// Sensor Settings
	fbSensor					: SH_Light.FB_NIKO_P46xx_1Pcs;
	//fbSensor					: SH_Light.FB_NIKO_P46xx_3Pcs;
	bySensorAddr				: BYTE := 1;
	//arrSensorAddr				: ARRAY[1..3] OF BYTE := [7,8,9];
	bInitialize					: BOOL := TRUE;
	stDaliSensorSetup			: ST_DALI_NIKOP46SetupData;
	bInitErr					: BOOL;
	bInitDone					: BOOL;
	//arrInitErr				: ARRAY [1..3] OF BOOL;
	//arrInitDone				: ARRAY [1..3] OF BOOL;
	arrSensorScales				: ARRAY [1..10] OF SH_Light.ST_DALI_SensorScaleMode := [
																						(fMeassureMaxSensor := rMeassure_Zone10, fReadMaxSensor := rRead_Zone10),																																									
																						9(())];
	bCancelHoldTimerOccupancy	: BOOL;
(*	eEventPriorityOccupancy		: E_DALIEventPriority := E_DALIEVENTPRIORITY.Middle;
	nHoldTimerOccupancy			: WORD := 5; // Value in s. 	
	nReportTimerOccupancy		: BYTE := 120; // Value in s, Preset manufacturer value
	nDeadtimeTimerOccupancy		: WORD := 100; // Value in ms, Predefined Value of DALI Standard
	bCancelHoldTimerOccupancy	: BOOL;
	nSensitivityOccupancy		: BYTE:= 3; //setting Sensivity (0..4) 0 (Off), 1 (Min), 2(Low), 3(High) and 4 (Max)

	bEnableLuxEvent				: BOOL;
	eEventPriorityBrightness	: E_DALIEventPriority := E_DALIEVENTPRIORITY.Middle;
	nDeadtimeTimerBrightness	: WORD := 1500; // Value in ms, Predefined Value of DALI Standard
	nHysteresisBrightness		: BYTE := 2; // Value in %
	nHysteresisMinBrightness	: BYTE := 10; // Absolute Value, depending on the manufacturer specific resolution
	nReportTimerBrightness		: BYTE := 120; // Value in s, Preset manufacturer value
*)

	//stDaliSetup: SH_Light.ST_DALI_RoomSetup
	//stRoomDataModbus			: SH_Light.ST_RoomDataModbus := ( bPirActive := bPirActive
	

	//ModbusComm setup
	
	fbWriteSPLuxLevel			: SH_Light.FB_TwoVal_SelectOne_RTrigChange;
	fbWritePirDelayTIme		: SH_Light.FB_TwoVal_SelectOne_RTrigChange;
	stRoomDataPLC				: SH_Light.ST_RoomDataPLC	:=	(
																	uiPirOffDelayTime	:= 30,
																	uiSpLuxLevel		:= 500,
																	uiPirDimDelayTime	:= 15,
																	uiSpDimLuxLevel		:= 200);
																	
	fbBallastOnHours				: SH_Light.FB_CountOnHours;
	bEnableHourCount			: BOOL := TRUE;
	
	//Non-persistent modbus data
	bPirActive_MB					AT %MX522.0	: BOOL;				//bPirLys i gammel kode
	uiActLuxLevel_MB			    AT %MB526	: UINT;				//intHMIAktueltLux i gammel kode
	uiActLightLevelPct_MB	        AT %MB530	: UINT;				//intDALI_Gruppe1_Lysniveau i gammel kode
	
	//For Conversion
	uiPirOffMinutes						: UINT;
	udTimeScaling						: UDINT := 60000;
	uiLuxOn								: UINT;
	
	//max values checks
	uiMaxLuxLevel						: UINT := 1023;
	uiMaxPirOffMinutes				    : UINT := 180;

	
END_VAR

VAR CONSTANT
    Sensor_DALI_LINE_NUM				: BYTE := 5;
	DALI_LINE_NUM_LIGHT			     	: BYTE := 2;
	DALI_LINE_NUM_PENDANTS	            : BYTE := 0; //0=ingen pendler	
END_VAR
VAR PERSISTENT
	stPirSensorData: SH_Light.ST_DALI_Sensor;
	stTuneData: SH_Light.ST_TuneData_EX;

	uiPirOffDelayTime_MB	AT %MB524	: UINT;				//ntHMI_Pir_SetValue i gammel kode
	uiSPLuxLevel_MB			AT %MB528	: UINT;				//intHMI_Lux_SetValue i gammel kode
	uiBallastOnHours_MB		AT %MB532	: UINT;				//dintHMILysbraendtimer1 i gammel kode
	byOnHoursOverflowCount				: BYTE;   
END_VAR

A_Buttons();
A_LightCtrl();
A_Sensor();
A_ModbusComm();

ACTION A_Buttons:
bTopButtonZone1		:= bTopButtonZone1_Visu;
bBottomButtonZone1	:= bBottomButtonZone1_Visu;
END_ACTION

ACTION A_LightCtrl:

fbLys(
	nZoneID:= 1, 
	bButtonZone1:= bTopButtonZone1,
	bBottomButtonZone1 := bBottomButtonZone1, 
	//bButtonZone2:= bButtonZone2,
	fLuxOn:= fLuxOn, 
	fLuxDim:= fLuxDim, 
	tPIRDim:= tPIRDim, 
	tPIROff:= tPIROff, 
	fOffsetSec:= fOffsetSec, 
	bReInit:= , 
	stDaliSetup:= stDaliSetup, 
	ipCommunication_Prim:= P_DALI_Background.arrfbKL6821Communication[DALI_LINE_NUM_LIGHT], 
	//ipCommunication_Sec:= P_DALI_Background.arrfbKL6821Communication[DALI_LINE_NUM_LIGHT], 
	//ipCommunication_Supl:= P_DALI_Background.arrfbKL6821Communication[DALI_LINE_NUM_PENDANTS], 
	fMinOutputPowerLevelRoom:= 15, 
	fMaxOutputPowerLevelRoom:= 100, 
	nCycleTimeInMS:= SH_Light.DALI_Param.nPlcTaskCycleTimeInMS*nDimCmdCycleTimeFactor , 
	bRunTuning:= bRunTuning, 
	bOccupiedRoom=> bOccupiedRoom, 
	bError_Prim=> , 
	nError_Prim=> , 
	stTuneData:=stTuneData , 
	stPirSensorData:= stPirSensorData, 
	stLiveData:= stLiveData);
END_ACTION

ACTION A_ModbusComm:
//Manage data for modbus communication

//Manage data for read-only in PLC
stRoomDataPLC.bPirActive			:= stPirSensorData.bPrc;
stRoomDataPLC.uiActLuxLevel			:= TO_UINT(TRUNC(stPirSensorData.fBrightness));
stRoomDataPLC.uiActLightLevelPct	:= TO_UINT(TRUNC(fbLys.fbBallast.fActlLgtLvl_Prim));
		//stRoomDataPLC.uiActLightLevelPct	:= TO_UINT(TRUNC(fbLys.fbBallast.fActlLgtLvl_Prim)); //if only one group light control
stRoomDataPLC.uiBallastOnHours		:= uiBallastOnHours_MB; //The calculation for BallastOnHours is stored directly to the MB register below


//Assign data for read-only to MB registers
bPirActive_MB			:= stRoomDataPLC.bPirActive;
uiActLuxLevel_MB		:= stRoomDataPLC.uiActLuxLevel;
uiActLightLevelPct_MB	:= stRoomDataPLC.uiActLightLevelPct;

	//calculate BallastOnHours
	fbBallastOnHours(
		bEnableHourCount	:= bEnableHourCount,
		bPauseCount			:= fbLys.fbLightCtrl.bOffZone1,
		uiOnHours			:= uiBallastOnHours_MB,			//OnHours is updated here
		byOverflowCount		:= byOnHoursOverflowCount);


//Manage data for read/write for both PLC and MB registers
fbWriteSPLuxLevel(	nMaxValOut	:= uiMaxLuxLevel,
					nValIn1		:= uiSPLuxLevel_MB,		//nValIn1 takes priotity in case of download or restart
					nValIn2		:= stRoomDataPLC.uiSpLuxLevel,
					nValOut		=> uiLuxOn
				);


fbWritePirDelayTIme(	nMaxValOut	:= uiMaxPirOffMinutes,
						nValIn1		:= uiPirOffDelayTime_MB,		//nValIn1 takes priotity in case of download or restart
						nValIn2		:= stRoomDataPLC.uiPirOffDelayTime,
						nValOut		=> uiPirOffMinutes
					);
					

//Convert read/write modbus data to appropriate datatypes in PLC
fLuxOn	:= TO_REAL(uiLuxOn);			
tPIROff	:= TO_TIME(uiPirOffMinutes*udTimeScaling); //Time conversion defaults to ms

fLuxDim	:= TO_REAL(stRoomDataPLC.uiSpDimLuxLevel);			
tPIRDim	:= TO_TIME(stRoomDataPLC.uiPirDimDelayTime*udTimeScaling); //Time conversion defaults to ms
END_ACTION

ACTION A_Sensor:

fbSensor.ipCommunication := P_DALI_Background.arrfbKL6821Communication[Sensor_DALI_LINE_NUM];

//only 1 sensor
fbSensor(
	byShrtAdr:= bySensorAddr,
	bInitialize:= bInitialize, 
	DALI_LINE_NUM:= Sensor_DALI_LINE_NUM, 
 	//bCancelHoldTimerOccupancy:= bCancelHoldTimerOccupancy, 
	stSensorSetup := stDaliSensorSetup,
	bInitErr=> bInitErr, 
	bInitDone=> bInitDone,
	stPirSensorData:= stPirSensorData, 
	arrSensorScales:= arrSensorScales);


(*//several sensors	
fbSensor(
	arrShrtAdr:= arrSensorAddr,
	bInitialize:= bInitialize, 
	DALI_LINE_NUM:= Sensor_DALI_LINE_NUM, 
 	//bCancelHoldTimerOccupancy:= bCancelHoldTimerOccupancy, 
	stSensorSetup := stDaliSensorSetup,
	arrInitErr=> arrInitErr, 
	arrInitDone=> arrInitDone,
	stPirSensorData:= stPirSensorData, 
	arrSensorScales:= arrSensorScales);
	*)
END_ACTION

END_PROGRAM

// ---- POUs/Alle_Rum/Gange/Gang_3_159A_toilet/P_Gang_3_159A.TcPOU
PROGRAM P_Gang_3_159A
VAR

	fbLys		: FB_Light_Type_B;
	

	stDaliSetup	: SH_Light.ST_DALI_RoomSetup := (
														byShrtAdr_Prim := 1, 
														byGrpAdr_Prim := 6,  /////remember
														eMod_Prim := E_DALIAddressType.Group, 
														//byShrtAdr_Sec := 1, 
														//byGrpAdr_Sec := 1, 
														//eMod_Sec := E_DALIAddressType.Short, 
														//byShrtAdr_Supl := 1, 
														DALI_LINE_NUM_PRIM := DALI_LINE_NUM_LIGHT,
														DALI_LINE_NUM_SEC := 0, //0 = ingen zonestyring/vinduerække
													    DALI_LINE_NUM_SUPL := DALI_LINE_NUM_PENDANTS);
														
	stLiveData				: SH_Light.ST_LiveData;
	bRunTuning					: BOOL;
	
	bTopButtonZone1				: BOOL;
	bTopButtonZone1_Visu		: BOOL;
	bBottomButtonZone1			: BOOL;
	bBottomButtonZone1_Visu	    : BOOL;
	bButtonZone2				: BOOL;
	bNeighborRoomsPir			: BOOL;
	fLuxOn						: REAL;
	fLuxDim						: REAL;
	tPIRDim						: TIME;
	tPIROff						: TIME;
	fOffsetSec					: REAL := 20;
	bOccupiedRoom				: BOOL;;


// Sensor Settings
	//fbSensor						: SH_Light.FB_NIKO_P46xx_1Pcs;
	fbSensor						: SH_Light.FB_NIKO_P46xx_2Pcs;
	//bySensorAddr				: BYTE := 1;
	arrSensorAddr				: ARRAY[1..2] OF BYTE := [4,5];
	bInitialize						: BOOL := TRUE;
	stDaliSensorSetup			: ST_DALI_NIKOP46SetupData := (
																nSensitivityPIRSegmentA := arrSensitivityOccupancy[1],
																nSensitivityPIRSegmentB := arrSensitivityOccupancy[2],
																nSensitivityPIRSegmentC := arrSensitivityOccupancy[3]);
	//bInitErr							: BOOL;
	//bInitDone						: BOOL;
	arrInitErr						: ARRAY [1..2] OF BOOL;
	arrInitDone					: ARRAY [1..2] OF BOOL;
	arrSensorScales				: ARRAY [1..10] OF SH_Light.ST_DALI_SensorScaleMode := [
																						(fMeassureMaxSensor := rMeassure_Zone10, fReadMaxSensor := rRead_Zone10),
																						(fMeassureMaxSensor := rMeassure_Zone10, fReadMaxSensor := rRead_Zone10),																																								
																						8(())];
																						
	bCancelHoldTimerOccupancy	: BOOL;
(*	eEventPriorityOccupancy		: E_DALIEventPriority := E_DALIEVENTPRIORITY.Middle;
	nHoldTimerOccupancy			: WORD := 5; // Value in s. 	
	nReportTimerOccupancy		: BYTE := 120; // Value in s, Preset manufacturer value
	nDeadtimeTimerOccupancy		: WORD := 100; // Value in ms, Predefined Value of DALI Standard
	bCancelHoldTimerOccupancy	: BOOL;
	nSensitivityOccupancy		: BYTE:= 3; //setting Sensivity (0..4) 0 (Off), 1 (Min), 2(Low), 3(High) and 4 (Max)

	bEnableLuxEvent				: BOOL;
	eEventPriorityBrightness	: E_DALIEventPriority := E_DALIEVENTPRIORITY.Middle;
	nDeadtimeTimerBrightness	: WORD := 1500; // Value in ms, Predefined Value of DALI Standard
	nHysteresisBrightness		: BYTE := 2; // Value in %
	nHysteresisMinBrightness	: BYTE := 10; // Absolute Value, depending on the manufacturer specific resolution
	nReportTimerBrightness		: BYTE := 120; // Value in s, Preset manufacturer value
*)
	

	//ModbusComm setup
	
	fbWriteSPLuxLevel				: SH_Light.FB_TwoVal_SelectOne_RTrigChange;
	fbWritePirDelayTIme			: SH_Light.FB_TwoVal_SelectOne_RTrigChange;
	stRoomDataPLC					: SH_Light.ST_RoomDataPLC	:=	(
																	uiPirOffDelayTime	:= 30,
																	uiSpLuxLevel			:= 500,
																	uiPirDimDelayTime	:= 15,
																	uiSpDimLuxLevel		:= 200);
																	
	fbBallastOnHours				: SH_Light.FB_CountOnHours;
	bEnableHourCount			: BOOL := TRUE;
	
	//Non-persistent modbus data
	bPirActive_MB				AT %MX534.0	: BOOL;				//bPirLys i gammel kode
	uiActLuxLevel_MB			AT %MB538	: UINT;				//intHMIAktueltLux i gammel kode
	uiActLightLevelPct_MB	    AT %MB542	: UINT;				//intDALI_Gruppe1_Lysniveau i gammel kode
	
	//For Conversion
	uiPirOffMinutes						: UINT;
	udTimeScaling						: UDINT := 60000;
	uiLuxOn								: UINT;
	
	//max values checks
	uiMaxLuxLevel						: UINT := 1023;
	uiMaxPirOffMinutes			    	: UINT := 180;

	
END_VAR

VAR CONSTANT
    Sensor_DALI_LINE_NUM				: BYTE := 4;
	DALI_LINE_NUM_LIGHT			    	: BYTE := 4;
	DALI_LINE_NUM_PENDANTS	            : BYTE := 0; //0=ingen pendler
	arrSensitivityOccupancy						: ARRAY[1..3] OF BYTE := [4,4,4];
END_VAR
VAR PERSISTENT
	stPirSensorData: SH_Light.ST_DALI_Sensor;
	stTuneData: SH_Light.ST_TuneData_EX;

	uiPirOffDelayTime_MB	AT %MB536	: UINT;				//ntHMI_Pir_SetValue i gammel kode
	uiSPLuxLevel_MB			AT %MB540	: UINT;				//intHMI_Lux_SetValue i gammel kode
	uiBallastOnHours_MB		AT %MB544	: UINT;				//dintHMILysbraendtimer1 i gammel kode
	byOnHoursOverflowCount							: BYTE;   
END_VAR

A_Buttons();
A_LightCtrl();
A_Sensor();
A_ModbusComm();

ACTION A_Buttons:
bTopButtonZone1		:= bTopButtonZone1_Visu;
bBottomButtonZone1	:= bBottomButtonZone1_Visu;
END_ACTION

ACTION A_LightCtrl:

fbLys(
	nZoneID:= 1, 
	bButtonZone1:= bTopButtonZone1,
	bBottomButtonZone1 := bBottomButtonZone1, 
	//bButtonZone2:= bButtonZone2, 
	bNeighborRoomsPir	:=	bNeighborRoomsPir,
	fLuxOn:= fLuxOn, 
	fLuxDim:= fLuxDim, 
	tPIRDim:= tPIRDim, 
	tPIROff:= tPIROff, 
	fOffsetSec:= fOffsetSec, 
	bReInit:= , 
	stDaliSetup:= stDaliSetup, 
	ipCommunication_Prim:= P_DALI_Background.arrfbKL6821Communication[DALI_LINE_NUM_LIGHT], 
	//ipCommunication_Sec:= P_DALI_Background.arrfbKL6821Communication[DALI_LINE_NUM_LIGHT], 
	//ipCommunication_Supl:= P_DALI_Background.arrfbKL6821Communication[DALI_LINE_NUM_PENDANTS], 
	fMinOutputPowerLevelRoom:= 15, 
	fMaxOutputPowerLevelRoom:= 100, 
	nCycleTimeInMS:= SH_Light.DALI_Param.nPlcTaskCycleTimeInMS*nDimCmdCycleTimeFactor , 
	bRunTuning:= bRunTuning, 
	bOccupiedRoom=> bOccupiedRoom, 
	bError_Prim=> , 
	nError_Prim=> , 
	stTuneData:=stTuneData , 
	stPirSensorData:= stPirSensorData, 
	stLiveData:= stLiveData);
END_ACTION

ACTION A_ModbusComm:
//Manage data for modbus communication

//Manage data for read-only in PLC
stRoomDataPLC.bPirActive			:= stPirSensorData.bPrc;
stRoomDataPLC.uiActLuxLevel			:= TO_UINT(TRUNC(stPirSensorData.fBrightness));
stRoomDataPLC.uiActLightLevelPct	:= TO_UINT(TRUNC(fbLys.fbBallast.fActlLgtLvl_Prim));
		//stRoomDataPLC.uiActLightLevelPct	:= TO_UINT(TRUNC(fbLys.fbBallast.fActlLgtLvl_Prim)); //if only one group light control
stRoomDataPLC.uiBallastOnHours		:= uiBallastOnHours_MB; //The calculation for BallastOnHours is stored directly to the MB register below


//Assign data for read-only to MB registers
bPirActive_MB			:= stRoomDataPLC.bPirActive;
uiActLuxLevel_MB		:= stRoomDataPLC.uiActLuxLevel;
uiActLightLevelPct_MB	:= stRoomDataPLC.uiActLightLevelPct;

	//calculate BallastOnHours
	fbBallastOnHours(
		bEnableHourCount	:= bEnableHourCount,
		bPauseCount			:= fbLys.fbLightCtrl.bOffZone1,
		uiOnHours			:= uiBallastOnHours_MB,			//OnHours is updated here
		byOverflowCount		:= byOnHoursOverflowCount);


//Manage data for read/write for both PLC and MB registers
fbWriteSPLuxLevel(	nMaxValOut	:= uiMaxLuxLevel,
					nValIn1		:= uiSPLuxLevel_MB,		//nValIn1 takes priotity in case of download or restart
					nValIn2		:= stRoomDataPLC.uiSpLuxLevel,
					nValOut		=> uiLuxOn
				);


fbWritePirDelayTIme(	nMaxValOut	:= uiMaxPirOffMinutes,
						nValIn1		:= uiPirOffDelayTime_MB,		//nValIn1 takes priotity in case of download or restart
						nValIn2		:= stRoomDataPLC.uiPirOffDelayTime,
						nValOut		=> uiPirOffMinutes
					);
					

//Convert read/write modbus data to appropriate datatypes in PLC
fLuxOn	:= TO_REAL(uiLuxOn);			
tPIROff	:= TO_TIME(uiPirOffMinutes*udTimeScaling); //Time conversion defaults to ms

fLuxDim	:= TO_REAL(stRoomDataPLC.uiSpDimLuxLevel);			
tPIRDim	:= TO_TIME(stRoomDataPLC.uiPirDimDelayTime*udTimeScaling); //Time conversion defaults to ms
END_ACTION

ACTION A_Sensor:

fbSensor.ipCommunication := P_DALI_Background.arrfbKL6821Communication[Sensor_DALI_LINE_NUM];

//only 1 sensor
(*fbSensor(
	byShrtAdr:= bySensorAddr,
	bInitialize:= bInitialize, 
	DALI_LINE_NUM:= Sensor_DALI_LINE_NUM, 
 	//bCancelHoldTimerOccupancy:= bCancelHoldTimerOccupancy, 
	stSensorSetup := stDaliSensorSetup,
	bInitErr=> bInitErr, 
	bInitDone=> bInitDone,
	stPirSensorData:= stPirSensorData, 
	arrSensorScales:= arrSensorScales);
*)

//several sensors	
fbSensor(
	arrShrtAdr:= arrSensorAddr,
	bInitialize:= bInitialize, 
	DALI_LINE_NUM:= Sensor_DALI_LINE_NUM, 
 	//bCancelHoldTimerOccupancy:= bCancelHoldTimerOccupancy, 
	stSensorSetup := stDaliSensorSetup,
	arrInitErr=> arrInitErr, 
	arrInitDone=> arrInitDone,
	stPirSensorData:= stPirSensorData, 
	arrSensorScales:= arrSensorScales);
END_ACTION

END_PROGRAM

// ---- POUs/Alle_Rum/Trapper/P_Trappe_T2.TcPOU
PROGRAM P_Trappe_T2
VAR
	bDigitalPir				AT%I*	: BOOL;
	bTrappelysNC		AT%Q*	: BOOL;
	

		
		
	fbTon_Off				: TON;
	tPirTidOff				: TIME;
	tPirTidOff_PLC	: TIME := T#1M;
	bIngenAktivitet		: BOOL;
	bTrappeLys			: BOOL;
	
	//Modbus data Read
	bTrappeAktivitet		: BOOL;
	//Modbus data Read/Wrtite
	bPirTidOff_MB			: TIME;
	
END_VAR


bIngenAktivitet	:= NOT bDigitalPir;
tPirTidOff		:= tPirTidOff_PLC;

fbTon_Off(IN:= bIngenAktivitet, PT:= tPirTidOff);

IF bDigitalPir  THEN
	bTrappeLys := TRUE;
END_IF
IF fbTon_Off.Q THEN
	bTrappeLys := FALSE;
END_IF

bTrappelysNC 	:= NOT bTrappeLys;

END_PROGRAM

// ---- POUs/Alle_Rum/Trapper/P_Trappe_T3.TcPOU
PROGRAM P_Trappe_T3
VAR
	bDigitalPir				AT%I*	: BOOL;
	bTrappelysNC		AT%Q*	: BOOL;
	

		
		
	fbTon_Off				: TON;
	tPirTidOff				: TIME;
	tPirTidOff_PLC	: TIME := T#1M;
	bIngenAktivitet		: BOOL;
	bTrappeLys			: BOOL;
	
	//Modbus data Read
	bTrappeAktivitet		: BOOL;
	//Modbus data Read/Wrtite
	bPirTidOff_MB			: TIME;
	
END_VAR


bIngenAktivitet	:= NOT bDigitalPir;
tPirTidOff		:= tPirTidOff_PLC;

fbTon_Off(IN:= bIngenAktivitet, PT:= tPirTidOff);

IF bDigitalPir  THEN
	bTrappeLys := TRUE;
END_IF
IF fbTon_Off.Q THEN
	bTrappeLys := FALSE;
END_IF

bTrappelysNC 	:= NOT bTrappeLys;

END_PROGRAM

// ---- POUs/DALI/DALI_Setup/FBs/FB_Part202Emergency.TcPOU
FUNCTION_BLOCK FB_Part202Emergency
VAR_INPUT
	ipDALICommunication					:	I_DALICommunication;
END_VAR
VAR_OUTPUT
	bBusy								:	BOOL;
END_VAR
VAR
	{region "Visu"}
	bReadCommands						:	BOOL;
	bReadState							:	BOOL;
	bReadParameter						:	BOOL;
	bStartFunctionTest					:	BOOL;
	bStopTest							:	BOOL;
	bStartDurationTest					:	BOOL;
	bResetFunctionTestDoneFlag			:	BOOL;
	bResetDurationTestDoneFlag			:	BOOL;
	bInhibit							:	BOOL;
	bResetInhibit						:	BOOL;
	bResetLampTime						:	BOOL;
	bRest								:	BOOL;
	bStartIdentification				:	BOOL;
	bWrite								:	BOOL;
	nBatteryCharge						:	BYTE;
	nDurationTestResult					:	BYTE;
	nLampEmergencyTime					:	BYTE;
	nLampTotalOperationTime				:	BYTE;
	sRestMode							:	STRING[5];
	sNormalMode							:	STRING[5];
	sEmergencyMode						:	STRING[5];
	sExtendedEmergency					:	STRING[5];
	sFunctionTest						:	STRING[5];
	sDurationTest						:	STRING[5];
	sHardwiredInhibit					:	STRING[5];
	sHardwiredSwitch					:	STRING[5];

	sCircuitFailure						:	STRING[5];
	sBatteryDurationFailure				:	STRING[5];
	sBatteryFailure						:	STRING[5];
	sEmergencyLampFailure				:	STRING[5];
	sFunctionTestExceed					:	STRING[5];
	sDurationTestExceed					:	STRING[5];
	sFunctionTestFailed					:	STRING[5];
	sDurationTestFailed					:	STRING[5];

	sInhibitMode						:	STRING[5];
	sFunctionTestDoneValid				:	STRING[5];
	sDurationTestDoneValid				:	STRING[5];
	sBatteryFullCharged					:	STRING[5];
	sFunctionTestRequestPending			:	STRING[5];
	sDurationTestRequestPending			:	STRING[5];
	sIdentificationActive				:	STRING[5];

	bIntegralControlGear				:	BOOL;
	bMaintainedControlGear				:	BOOL;
	bSwitchtedMaintainedControlGear		:	BOOL;
	bAutoTestCapability					:	BOOL;
	bAdjustableEmergencyLevel			:	BOOL;
	bHardwiredInhibitSupported			:	BOOL;
	bPhysicalSelectionSupported			:	BOOL;
	bRelightinRestModeSupported			:	BOOL;

	nEmergencyLevel						:	BYTE;
	nEmergencyMinLevel					:	BYTE;
	nEmergencyMaxLevel					:	BYTE;
	nProlongTime						:	UINT;
	fDurationTestDelayTimeVisu			:	REAL;
	fFunctionTestDelayTimeVisu			:	REAL;
	nFunctionTestInterval				:	UINT;
	nDurationTestInterval				:	UINT;
	nTestExecutionTimeout				:	UINT;
	nRatedDuration						:	BYTE;
	{endregion}
	nStep								:	INT;
	nAddress							:	BYTE;
	bHideWaitSymbol						:	BOOL := TRUE;
	
	nDurationTestDelayTime				:	UINT;
	nFunctionTestDelayTime				:	UINT;
	
	fb103StartQuiescentMode				:	FB_DALI103StartQuiescentMode(0);
	fb103StopQuiescentMode				:	FB_DALI103StopQuiescentMode(0);
	fb202QueryBatteryCharge				:	FB_DALI202QueryBatteryCharge(0);
	fb202QueryDurationTestResult		:	FB_DALI202QueryDurationTestResult(0);
	fb202QueryLampEmergencyTime			:	FB_DALI202QueryLampEmergencyTime(0);
	fb202QueryLampTotalOperationTime	:	FB_DALI202QueryLampTotalOperationTime(0);
	fb202QueryEmergencyLevel			:	FB_DALI202QueryEmergencyLevel(0);
	fb202QueryEmergencyMode				:	FB_DALI202QueryEmergencyMode(0);
	fb202QueryFailureStatus				:	FB_DALI202QueryFailureStatus(0);
	fb202QueryEmergencyStatus			:	FB_DALI202QueryEmergencyStatus(0);
	
	fb202QueryEmergencyMinLevel			:	FB_DALI202QueryEmergencyMinLevel(0);
	fb202QueryEmergencyMaxLevel			:	FB_DALI202QueryEmergencyMaxLevel(0);
	fb202QueryTestTiming				:	FB_DALI202QueryTestTiming(0);
	fb202QueryRatedDuration				:	FB_DALI202QueryRatedDuration(0);
	fb202QueryFeatures					:	FB_DALI202QueryFeatures(0);
	
	fb202SetEmergencyLevel				:	FB_DALI202SetEmergencyLevel(0);
	fb202SetProlongTime					:	FB_DALI202SetProlongTime(0);
	fb202SetTestDelayTime				:	FB_DALI202SetTestDelayTime(0);
	fb202SetFunctionTestInterval		:	FB_DALI202SetFunctionTestInterval(0);
	fb202SetDurationTestInterval		:	FB_DALI202SetDurationTestInterval(0);
	fb202SetTestExecutionTimeout		:	FB_DALI202SetTestExecutionTimeout(0);
	
	fb202StartFunctionTest				:	FB_DALI202StartFunctionTest(0);
	fb202StopTest						:	FB_DALI202StopTest(0);
	fb202StartDurationTest				:	FB_DALI202StartDurationTest(0);
	fb202ResetFunctionTestDoneFlag		:	FB_DALI202ResetFunctionTestDoneFlag(0);
	fb202ResetDurationTestDoneFlag		:	FB_DALI202ResetDurationTestDoneFlag(0);
	fb202Inhibit						:	FB_DALI202Inhibit(0);
	fb202ReLightResetInhibit			:	FB_DALI202ReLightResetInhibit(0);
	fb202ResetLampTime					:	FB_DALI202ResetLampTime(0);
	fb202Rest							:	FB_DALI202Rest(0);
	fb202StartIdentification			:	FB_DALI202StartIdentification(0);
END_VAR

{region "Detect Commands"}
IF (bStartFunctionTest AND (nStep = 0)) THEN
	nStep := 5;
	bStartFunctionTest := FALSE;
END_IF

IF (bStopTest AND (nStep = 0)) THEN
	nStep := 10;
	bStopTest := FALSE;
END_IF

IF (bStartDurationTest AND (nStep = 0)) THEN
	nStep := 15;
	bStartDurationTest := FALSE;
END_IF

IF (bResetFunctionTestDoneFlag AND (nStep = 0)) THEN
	nStep := 20;
	bResetFunctionTestDoneFlag := FALSE;
END_IF

IF (bResetDurationTestDoneFlag AND (nStep = 0)) THEN
	nStep := 25;
	bResetDurationTestDoneFlag := FALSE;
END_IF

IF (bInhibit AND (nStep = 0)) THEN
	nStep := 30;
	bInhibit := FALSE;
END_IF

IF (bResetInhibit AND (nStep = 0)) THEN
	nStep := 35;
	bResetInhibit := FALSE;
END_IF

IF (bResetLampTime AND (nStep = 0)) THEN
	nStep := 40;
	bResetLampTime := FALSE;
END_IF			   
					
IF (bRest AND (nStep = 0)) THEN
	nStep := 45;
	bRest := FALSE;
END_IF

IF (bStartIdentification AND (nStep = 0)) THEN
	nStep := 50;
	bStartIdentification := FALSE;
END_IF

IF (bReadCommands AND (nStep = 0)) THEN
	nStep := 60;
	bReadCommands := FALSE;
	bHideWaitSymbol := FALSE;
END_IF

IF (bReadState AND (nStep = 0)) THEN
	nStep := 100;
	bReadState := FALSE;
	bHideWaitSymbol := FALSE;
END_IF

IF (bReadParameter AND (nStep = 0)) THEN
	nStep := 200;
	bReadParameter := FALSE;
	bHideWaitSymbol := FALSE;
END_IF

IF (bWrite AND (nStep = 0)) THEN
	nStep := 500;
	bWrite := FALSE;
	bHideWaitSymbol := FALSE;
END_IF
{endregion}
{region "Manage Dialog Selection}
IF (nStep = 0) THEN
	bBusy := FALSE;
ELSE
	bBusy := TRUE;
END_IF
{endregion}
{region "Execute Commands"}
CASE nStep OF
0:
{region "Init"}
	bReadCommands := FALSE;
	bReadState := FALSE;
	bReadParameter := FALSE;
	bWrite := FALSE;
	bHideWaitSymbol := TRUE;

	fb103StartQuiescentMode.ipDALICommunication := ipDALICommunication;
	fb103StopQuiescentMode.ipDALICommunication := ipDALICommunication;
	fb202QueryBatteryCharge.ipDALICommunication := ipDALICommunication;
	fb202QueryDurationTestResult.ipDALICommunication := ipDALICommunication;
	fb202QueryDurationTestResult.ipDALICommunication := ipDALICommunication;
	fb202QueryLampEmergencyTime.ipDALICommunication := ipDALICommunication;
	fb202QueryLampTotalOperationTime.ipDALICommunication := ipDALICommunication;
	fb202QueryEmergencyMode.ipDALICommunication := ipDALICommunication;
	fb202QueryFailureStatus.ipDALICommunication := ipDALICommunication;
	fb202QueryEmergencyStatus.ipDALICommunication := ipDALICommunication;
	fb202QueryEmergencyLevel.ipDALICommunication := ipDALICommunication;
	fb202QueryEmergencyMinLevel.ipDALICommunication := ipDALICommunication;
	fb202QueryEmergencyMaxLevel.ipDALICommunication := ipDALICommunication;
	fb202QueryTestTiming.ipDALICommunication := ipDALICommunication;
	fb202QueryRatedDuration.ipDALICommunication := ipDALICommunication;
	fb202QueryFeatures.ipDALICommunication := ipDALICommunication;
	fb202SetEmergencyLevel.ipDALICommunication := ipDALICommunication;
	fb202SetProlongTime.ipDALICommunication := ipDALICommunication;
	fb202SetTestDelayTime.ipDALICommunication := ipDALICommunication;
	fb202SetFunctionTestInterval.ipDALICommunication := ipDALICommunication;
	fb202SetDurationTestInterval.ipDALICommunication := ipDALICommunication;
	fb202SetTestExecutionTimeout.ipDALICommunication := ipDALICommunication;

	fb202StartFunctionTest.ipDALICommunication := ipDALICommunication;
	fb202StopTest.ipDALICommunication := ipDALICommunication;
	fb202StartDurationTest.ipDALICommunication := ipDALICommunication;
	fb202ResetFunctionTestDoneFlag.ipDALICommunication := ipDALICommunication;
	fb202ResetDurationTestDoneFlag.ipDALICommunication := ipDALICommunication;
	fb202Inhibit.ipDALICommunication := ipDALICommunication;
	fb202ReLightResetInhibit.ipDALICommunication := ipDALICommunication;
	fb202ResetLampTime.ipDALICommunication := ipDALICommunication;
	fb202Rest.ipDALICommunication := ipDALICommunication;
	fb202StartIdentification.ipDALICommunication := ipDALICommunication;
{endregion}
{region "Commands"}
5:
	fb202StartFunctionTest(	bStart:= TRUE,
							nAddress := nAddress,
							eAddressType := Tc3_DALI.E_DALIAddressType.Short,
							eCommandPriority := Tc3_DALI.E_DALICommandPriority.Middle);
	IF (NOT fb202StartFunctionTest.bBusy) THEN
		fb202StartFunctionTest(bStart := FALSE);
		nStep :=0;
	END_IF
10:
	fb202StopTest(	bStart:= TRUE,
					nAddress := nAddress,
					eAddressType := Tc3_DALI.E_DALIAddressType.Short,
					eCommandPriority := Tc3_DALI.E_DALICommandPriority.Middle);
	IF (NOT fb202StopTest.bBusy) THEN
		fb202StopTest(bStart := FALSE);
		nStep :=0;
	END_IF
15:
	fb202StartDurationTest(	bStart:= TRUE,
							nAddress := nAddress,
							eAddressType := Tc3_DALI.E_DALIAddressType.Short,
							eCommandPriority := Tc3_DALI.E_DALICommandPriority.Middle);
	IF (NOT fb202StartDurationTest.bBusy) THEN
		fb202StartDurationTest(bStart := FALSE);
		nStep := 0;
	END_IF
20:
	fb202ResetFunctionTestDoneFlag(	bStart := TRUE,
									nAddress := nAddress,
									eAddressType := Tc3_DALI.E_DALIAddressType.Short,
									eCommandPriority := Tc3_DALI.E_DALICommandPriority.Middle);
	IF (NOT fb202ResetFunctionTestDoneFlag.bBusy) THEN
		fb202ResetFunctionTestDoneFlag(bStart := FALSE);
		nStep := 0;
	END_IF
25:
	fb202ResetDurationTestDoneFlag(	bStart:= TRUE,
									nAddress := nAddress,
									eAddressType := Tc3_DALI.E_DALIAddressType.Short,
									eCommandPriority := Tc3_DALI.E_DALICommandPriority.Middle);
	IF (NOT fb202ResetDurationTestDoneFlag.bBusy) THEN
		fb202ResetDurationTestDoneFlag(bStart := FALSE);
		nStep := 0;
	END_IF
30:
	fb202Inhibit(	bStart := TRUE,
					nAddress := nAddress,
					eAddressType := Tc3_DALI.E_DALIAddressType.Short,
					eCommandPriority := Tc3_DALI.E_DALICommandPriority.Middle);
	IF (NOT fb202Inhibit.bBusy) THEN
		fb202Inhibit(bStart := FALSE);
		nStep := 0;
	END_IF
35:
	fb202ReLightResetInhibit(	bStart := TRUE,
								nAddress := nAddress,
								eAddressType := Tc3_DALI.E_DALIAddressType.Short,
								eCommandPriority := Tc3_DALI.E_DALICommandPriority.Middle);
	IF (NOT fb202ReLightResetInhibit.bBusy) THEN
		fb202ReLightResetInhibit(bStart := FALSE);
		nStep := 0;
	END_IF
40:
	fb202ResetLampTime(	bStart := TRUE,
						nAddress := nAddress,
						eAddressType := Tc3_DALI.E_DALIAddressType.Short,
						eCommandPriority := Tc3_DALI.E_DALICommandPriority.Middle);
	IF (NOT fb202ResetLampTime.bBusy) THEN
		fb202ResetLampTime(bStart := FALSE);
		nStep := 0;
	END_IF
45:
	fb202Rest(	bStart := TRUE,
				nAddress := nAddress,
				eAddressType := Tc3_DALI.E_DALIAddressType.Short,
				eCommandPriority := Tc3_DALI.E_DALICommandPriority.Middle);
	IF (NOT fb202Rest.bBusy) THEN
		fb202Rest(bStart := FALSE);
		nStep := 0;
	END_IF
50:
	fb202StartIdentification(	bStart := TRUE,
								nAddress := nAddress,
								eAddressType := Tc3_DALI.E_DALIAddressType.Short,
								eCommandPriority := Tc3_DALI.E_DALICommandPriority.Middle);
	IF (NOT fb202StartIdentification.bBusy) THEN
		fb202StartIdentification(bStart := FALSE);
		nStep := 0;
	END_IF
{endregion}
{region "Read Command Status"}
55:
{region "Start Qiescent Mode"}
	fb103StartQuiescentMode(bStart := TRUE,
							eAddressType := Tc3_DALI.E_DALIAddressType.Broadcast,
							eCommandPriority := Tc3_DALI.E_DALICommandPriority.Middle);
	IF (NOT fb103StartQuiescentMode.bBusy) THEN
		fb103StartQuiescentMode(bStart := FALSE);
		nStep := 60;
	END_IF
{endregion}
{endregion}
60:
{region "Query Battery Charge"}
	fb202QueryBatteryCharge(bStart := TRUE,
							nAddress := nAddress,
							eAddressType := Tc3_DALI.E_DALIAddressType.Short,
							eCommandPriority := Tc3_DALI.E_DALICommandPriority.Middle );
	IF (NOT fb202QueryBatteryCharge.bBusy) THEN
		fb202QueryBatteryCharge(bStart:= FALSE);
		nBatteryCharge := fb202QueryBatteryCharge.nBatteryCharge;
		nStep := 65;
	END_IF
{endregion}
65:
{region "Query Duration Test Result"}
	fb202QueryDurationTestResult(	bStart := TRUE,
									nAddress := nAddress,
									eAddressType := Tc3_DALI.E_DALIAddressType.Short,
									eCommandPriority := Tc3_DALI.E_DALICommandPriority.Middle );
	IF (NOT fb202QueryDurationTestResult.bBusy) THEN
		fb202QueryDurationTestResult(bStart := FALSE);
		nDurationTestResult := (2 * fb202QueryDurationTestResult.nDurationTestResult);
		nStep := 70;
	END_IF
{endregion}
70:
{region "Query Lamp emergency Time"}
	fb202QueryLampEmergencyTime(	bStart := TRUE,
									nAddress := nAddress,
									eAddressType := Tc3_DALI.E_DALIAddressType.Short,
									eCommandPriority := Tc3_DALI.E_DALICommandPriority.Middle );
	IF (NOT fb202QueryLampEmergencyTime.bBusy) THEN
		fb202QueryLampEmergencyTime(bStart := FALSE);
		nLampEmergencyTime := fb202QueryLampEmergencyTime.nLampEmergencyTime;
		nStep := 75;
	END_IF
{endregion}
75:
{region "Query Lamp total operation Time"}
	fb202QueryLampTotalOperationTime(	bStart := TRUE,
										nAddress := nAddress,
										eAddressType := Tc3_DALI.E_DALIAddressType.Short,
										eCommandPriority := Tc3_DALI.E_DALICommandPriority.Middle );
	IF (NOT fb202QueryLampTotalOperationTime.bBusy) THEN
		fb202QueryLampTotalOperationTime(bStart:= FALSE);
		nLampTotalOperationTime := (4 * fb202QueryLampTotalOperationTime.nLampTotalOperationTime);
		nStep := 80;
	END_IF
{endregion}
80:
{region "Stop Quiescent Mode"}
	fb103StopQuiescentMode(bStart := TRUE,
							eAddressType := Tc3_DALI.E_DALIAddressType.Broadcast,
							eCommandPriority := Tc3_DALI.E_DALICommandPriority.Middle);
	IF (NOT fb103StopQuiescentMode.bBusy) THEN
		fb103StopQuiescentMode(bStart := FALSE);
		nStep := 0;
	END_IF
	{endregion}

{region "Read Status"}
100:
{region "Query Emergency Mode"}
	fb202QueryEmergencyMode(bStart := TRUE,
							nAddress := nAddress,
							eAddressType := Tc3_DALI.E_DALIAddressType.Short,
							eCommandPriority := Tc3_DALI.E_DALICommandPriority.Middle );
	IF (NOT fb202QueryEmergencyMode.bBusy) THEN
		fb202QueryEmergencyMode(bStart:= FALSE);
		sRestMode := SEL(fb202QueryEmergencyMode.nEmergencyMode.0, 'FALSE', 'TRUE');
		sNormalMode := SEL(fb202QueryEmergencyMode.nEmergencyMode.1, 'FALSE', 'TRUE');
		sEmergencyMode := SEL(fb202QueryEmergencyMode.nEmergencyMode.2, 'FALSE', 'TRUE');
		sExtendedEmergency := SEL(fb202QueryEmergencyMode.nEmergencyMode.3, 'FALSE', 'TRUE');
		sFunctionTest := SEL(fb202QueryEmergencyMode.nEmergencyMode.4, 'FALSE', 'TRUE');
		sDurationTest := SEL(fb202QueryEmergencyMode.nEmergencyMode.5, 'FALSE', 'TRUE');
		sHardwiredInhibit := SEL(fb202QueryEmergencyMode.nEmergencyMode.6, 'FALSE', 'TRUE');
		sHardwiredSwitch := SEL(fb202QueryEmergencyMode.nEmergencyMode.7, 'FALSE', 'TRUE');
		nStep := 110;
	END_IF
{endregion}
110:
{region "Query Failure Status"}
	fb202QueryFailureStatus(bStart := TRUE,
							nAddress := nAddress,
							eAddressType := Tc3_DALI.E_DALIAddressType.Short,
							eCommandPriority := Tc3_DALI.E_DALICommandPriority.Middle );
	IF (NOT fb202QueryFailureStatus.bBusy) THEN
		fb202QueryFailureStatus(bStart := FALSE);
		sCircuitFailure := SEL(fb202QueryFailureStatus.nFailureStatus.0, 'FALSE', 'TRUE');
		sBatteryDurationFailure := SEL(fb202QueryFailureStatus.nFailureStatus.1, 'FALSE', 'TRUE');
		sBatteryFailure := SEL(fb202QueryFailureStatus.nFailureStatus.2, 'FALSE', 'TRUE');
		sEmergencyLampFailure := SEL(fb202QueryFailureStatus.nFailureStatus.3, 'FALSE', 'TRUE');
		sFunctionTestExceed := SEL(fb202QueryFailureStatus.nFailureStatus.4, 'FALSE', 'TRUE');
		sDurationTestExceed := SEL(fb202QueryFailureStatus.nFailureStatus.5, 'FALSE', 'TRUE');
		sFunctionTestFailed := SEL(fb202QueryFailureStatus.nFailureStatus.6, 'FALSE', 'TRUE');
		sDurationTestFailed := SEL(fb202QueryFailureStatus.nFailureStatus.7, 'FALSE', 'TRUE');
		nStep := 120;
	END_IF
{endregion}
120:
{region "Query Emergency Status"}
	fb202QueryEmergencyStatus(bStart := TRUE,
							nAddress := nAddress,
							eAddressType := Tc3_DALI.E_DALIAddressType.Short,
							eCommandPriority := Tc3_DALI.E_DALICommandPriority.Middle );
	IF (NOT fb202QueryEmergencyStatus.bBusy) THEN
		fb202QueryEmergencyStatus(bStart := FALSE);
		sInhibitMode := SEL(fb202QueryEmergencyStatus.nEmergencyStatus.0, 'FALSE', 'TRUE');
		sFunctionTestDoneValid := SEL(fb202QueryEmergencyStatus.nEmergencyStatus.1, 'FALSE', 'TRUE');
		sDurationTestDoneValid := SEL(fb202QueryEmergencyStatus.nEmergencyStatus.2, 'FALSE', 'TRUE');
		sBatteryFullCharged := SEL(fb202QueryEmergencyStatus.nEmergencyStatus.3, 'FALSE', 'TRUE');
		sFunctionTestRequestPending := SEL(fb202QueryEmergencyStatus.nEmergencyStatus.4, 'FALSE', 'TRUE');
		sDurationTestRequestPending := SEL(fb202QueryEmergencyStatus.nEmergencyStatus.5, 'FALSE', 'TRUE');
		sIdentificationActive := SEL(fb202QueryEmergencyStatus.nEmergencyStatus.6, 'FALSE', 'TRUE');
		nStep := 0;
	END_IF
{endregion}
{endregion}
{region "Read Parameters"}
200:
	{region "Start Qiescent Mode"}
	fb103StartQuiescentMode(bStart := TRUE,
							eAddressType := Tc3_DALI.E_DALIAddressType.Broadcast,
							eCommandPriority := Tc3_DALI.E_DALICommandPriority.Middle);
	IF (NOT fb103StartQuiescentMode.bBusy) THEN
		fb103StartQuiescentMode(bStart := FALSE);
		nStep := 210;
	END_IF
{endregion}
210:
{region "Query Emergency Level"}
	fb202QueryEmergencyLevel(	bStart := TRUE,
								nAddress := nAddress,
								eAddressType := Tc3_DALI.E_DALIAddressType.Short,
								eCommandPriority := Tc3_DALI.E_DALICommandPriority.Middle );
	IF (NOT fb202QueryEmergencyLevel.bBusy) THEN
		fb202QueryEmergencyLevel (bStart := FALSE);
		nEmergencyLevel := fb202QueryEmergencyLevel.nEmergencyLevel;
		nStep := 220;
	END_IF
{endregion}
220:
{region "Query Emergency Min Level"}
	fb202QueryEmergencyMinLevel(bStart := TRUE,
								nAddress := nAddress,
								eAddressType := Tc3_DALI.E_DALIAddressType.Short,
								eCommandPriority := Tc3_DALI.E_DALICommandPriority.Middle );
	IF (NOT fb202QueryEmergencyMinLevel.bBusy) THEN
		fb202QueryEmergencyMinLevel (bStart := FALSE);
		nEmergencyMinLevel := fb202QueryEmergencyMinLevel.nEmergencyMinLevel;
		nStep := 230;
	END_IF
{endregion}
230:
{region "Query Emergency Max Level"}
	fb202QueryEmergencyMaxLevel(bStart := TRUE,
								nAddress := nAddress,
								eAddressType := Tc3_DALI.E_DALIAddressType.Short,
								eCommandPriority := Tc3_DALI.E_DALICommandPriority.Middle );
	IF (NOT fb202QueryEmergencyMaxLevel.bBusy) THEN
		fb202QueryEmergencyMaxLevel (bStart := FALSE);
		nEmergencyMaxLevel := fb202QueryEmergencyMaxLevel.nEmergencyMaxLevel;
		nStep := 240;
	END_IF
{endregion}
240: 
{region "Query Prolong Time"}
	fb202QueryTestTiming(	bStart := TRUE,
							nAddress := nAddress,
							eAddressType := Tc3_DALI.E_DALIAddressType.Short,
							eCommandPriority := Tc3_DALI.E_DALICommandPriority.Middle,
							eTestTiming:= Tc3_DALI.E_DALITestTiming.ProlongTime);
	IF (NOT fb202QueryTestTiming.bBusy) THEN
		fb202QueryTestTiming (bStart := FALSE);
		nProlongTime := (fb202QueryTestTiming.nValue * 30);
		nStep := 250;
	END_IF
{endregion}
250:
{region "Query Function Test Delay Time"}
	fb202QueryTestTiming(	bStart := TRUE,
							nAddress := nAddress,
							eAddressType := Tc3_DALI.E_DALIAddressType.Short,
							eCommandPriority := Tc3_DALI.E_DALICommandPriority.Middle,
							eTestTiming:= Tc3_DALI.E_DALITestTiming.FunctionTestDelayTime );
	IF (NOT fb202QueryTestTiming.bBusy) THEN
		fb202QueryTestTiming (bStart := FALSE);
		nFunctionTestDelayTime := (fb202QueryTestTiming.nValue * 15);
		fFunctionTestDelayTimeVisu := TO_REAL(nFunctionTestDelayTime)/ 60;
		nStep := 260;
	END_IF
{endregion}
260:
{region "Query Duration Test Delay Time"}
	fb202QueryTestTiming(	bStart := TRUE,
							nAddress := nAddress,
							eAddressType := Tc3_DALI.E_DALIAddressType.Short,
							eCommandPriority := Tc3_DALI.E_DALICommandPriority.Middle,
							eTestTiming := Tc3_DALI.E_DALITestTiming.DurationTestDelayTime);
	IF (NOT fb202QueryTestTiming.bBusy) THEN
		fb202QueryTestTiming (bStart := FALSE);
		nDurationTestDelayTime := (fb202QueryTestTiming.nValue * 15);
		fDurationTestDelayTimeVisu := TO_REAL(nDurationTestDelayTime) / 60;
		nStep := 270;
	END_IF
{endregion}
270:
{region "Query Function Test Interval"}
	fb202QueryTestTiming(	bStart := TRUE,
							nAddress := nAddress,
							eAddressType := Tc3_DALI.E_DALIAddressType.Short,
							eCommandPriority := Tc3_DALI.E_DALICommandPriority.Middle,
							eTestTiming:= Tc3_DALI.E_DALITestTiming.FunctionTestInterval);
	IF (NOT fb202QueryTestTiming.bBusy) THEN
		fb202QueryTestTiming (bStart := FALSE);
		nFunctionTestInterval := fb202QueryTestTiming.nValue;
		nStep := 280;
	END_IF
{endregion}
280:
{region "Query Duration Test Interval"}
	fb202QueryTestTiming(	bStart := TRUE,
							nAddress := nAddress,
							eAddressType := Tc3_DALI.E_DALIAddressType.Short,
							eCommandPriority := Tc3_DALI.E_DALICommandPriority.Middle,
							eTestTiming:= Tc3_DALI.E_DALITestTiming.DurationTestInterval);
	IF (NOT fb202QueryTestTiming.bBusy) THEN
		fb202QueryTestTiming (bStart := FALSE);
		nDurationTestInterval := fb202QueryTestTiming.nValue;
		nStep := 290;
	END_IF
{endregion}
290:
{region "Query Test Execution Timeout"}
	fb202QueryTestTiming(	bStart := TRUE,
							nAddress := nAddress,
							eAddressType := Tc3_DALI.E_DALIAddressType.Short,
							eCommandPriority := Tc3_DALI.E_DALICommandPriority.Middle,
							eTestTiming:= Tc3_DALI.E_DALITestTiming.TestExecutionTimeout);
	IF (NOT fb202QueryTestTiming.bBusy) THEN
		fb202QueryTestTiming (bStart := FALSE);
		nTestExecutionTimeout := fb202QueryTestTiming.nValue;
		nStep := 300;
	END_IF
{endregion}
300:
{region "Query Rated Duration"}
	fb202QueryRatedDuration(bStart := TRUE,
							nAddress := nAddress,
							eAddressType := Tc3_DALI.E_DALIAddressType.Short,
							eCommandPriority := Tc3_DALI.E_DALICommandPriority.Middle );
	IF (NOT fb202QueryRatedDuration.bBusy) THEN
		fb202QueryRatedDuration (bStart := FALSE);
		nRatedDuration := ( 2 * fb202QueryRatedDuration.nRatedDuration);
		nStep := 310;
	END_IF
{endregion}
310:
{region "Query Features"}
	fb202QueryFeatures(	bStart := TRUE,
						nAddress := nAddress,
						eAddressType := Tc3_DALI.E_DALIAddressType.Short,
						eCommandPriority := Tc3_DALI.E_DALICommandPriority.Middle );
	IF (NOT fb202QueryFeatures.bBusy) THEN
		fb202QueryFeatures (bStart := FALSE);
		bIntegralControlGear	:= fb202QueryFeatures.nFeatures.0;
		bMaintainedControlGear	:= fb202QueryFeatures.nFeatures.1;
		bSwitchtedMaintainedControlGear	:= fb202QueryFeatures.nFeatures.2;
		bAutoTestCapability	:= fb202QueryFeatures.nFeatures.3;
		bAdjustableEmergencyLevel	:= fb202QueryFeatures.nFeatures.4;
		bHardwiredInhibitSupported	:= fb202QueryFeatures.nFeatures.5;
		bPhysicalSelectionSupported	:= fb202QueryFeatures.nFeatures.6;
		bRelightinRestModeSupported	:= fb202QueryFeatures.nFeatures.7;
		nStep := 320;
	END_IF
{endregion}
320:
{region "Stop Quiescent Mode"}
	 fb103StopQuiescentMode(bStart := TRUE,
							eAddressType := Tc3_DALI.E_DALIAddressType.Broadcast,
							eCommandPriority := Tc3_DALI.E_DALICommandPriority.Middle);
	IF (NOT fb103StopQuiescentMode.bBusy) THEN
		fb103StopQuiescentMode(bStart := FALSE);
		nStep := 0;
	END_IF
{endregion}
{endregion}
{region "Write Parameters"}
500:
{region "Set Emergency Level"}
	fb202SetEmergencyLevel(	bStart := TRUE,
							nAddress := nAddress,
							eAddressType := Tc3_DALI.E_DALIAddressType.Short,
							eCommandPriority := Tc3_DALI.E_DALICommandPriority.Middle,
							nEmergencyLevel :=  nEmergencyLevel);
	IF (NOT fb202SetEmergencyLevel.bBusy) THEN
		fb202SetEmergencyLevel (bStart := FALSE);
		nStep := 510;
	END_IF
{endregion}
510:
{region "Set Prolong Time"}
	fb202SetProlongTime(	bStart := TRUE,
							nAddress := nAddress,
							eAddressType := Tc3_DALI.E_DALIAddressType.Short,
							eCommandPriority := Tc3_DALI.E_DALICommandPriority.Middle,
							nProlongTime:= TO_BYTE(nProlongTime / 30));
	IF (NOT fb202SetProlongTime.bBusy) THEN
		fb202SetProlongTime (bStart := FALSE);
		nStep := 520;
	END_IF
{endregion}
520:
	nDurationTestDelayTime := TO_UINT((fDurationTestDelayTimeVisu *60) /15);
	fb202SetTestDelayTime(	bStart := TRUE,
							nAddress := nAddress,
							eAddressType := Tc3_DALI.E_DALIAddressType.Short,
							eCommandPriority := Tc3_DALI.E_DALICommandPriority.Middle,
							nTestDelayTime := nDurationTestDelayTime);
	IF (NOT fb202SetTestDelayTime.bBusy) THEN
		fb202SetTestDelayTime (bStart := FALSE);
		nStep := 530;
	END_IF
530:
	fb202SetDurationTestInterval(	bStart := TRUE,
									nAddress := nAddress,
									eAddressType := Tc3_DALI.E_DALIAddressType.Short,
									eCommandPriority := Tc3_DALI.E_DALICommandPriority.Middle,
									nDurationTestInterval := TO_BYTE(nDurationTestInterval));
	IF (NOT fb202SetDurationTestInterval.bBusy) THEN
		fb202SetDurationTestInterval(bStart := FALSE);
		nStep := 540;
	END_IF
{endregion}
{region "Set Function Test Delay time and Function Test Interval"}
540:
	nFunctionTestDelayTime := TO_UINT(fFunctionTestDelayTimeVisu * 60 / 15);
	fb202SetTestDelayTime(	bStart := TRUE,
							nAddress := nAddress,
							eAddressType := Tc3_DALI.E_DALIAddressType.Short,
							eCommandPriority := Tc3_DALI.E_DALICommandPriority.Middle,
							nTestDelayTime := nFunctionTestDelayTime);
	IF (NOT fb202SetTestDelayTime.bBusy) THEN
		fb202SetTestDelayTime(bStart := FALSE);
		nStep := 550;
	END_IF
550:
	fb202SetFunctionTestInterval(	bStart := TRUE,
									nAddress := nAddress,
									eAddressType := Tc3_DALI.E_DALIAddressType.Short,
									eCommandPriority := Tc3_DALI.E_DALICommandPriority.Middle,
									nFunctionTestInterval := TO_BYTE(nFunctionTestInterval));
	IF (NOT fb202SetFunctionTestInterval.bBusy) THEN
		fb202SetFunctionTestInterval (bStart := FALSE);
		nStep := 560;
	END_IF
{endregion}
560:
{region "Set Test Execution Timeout"}
	fb202SetTestExecutionTimeout(	bStart := TRUE,
									nAddress := nAddress,
									eAddressType := Tc3_DALI.E_DALIAddressType.Short,
									eCommandPriority := Tc3_DALI.E_DALICommandPriority.Middle,
									nTestExecutionTimeout := TO_BYTE(nTestExecutionTimeout));
	IF (NOT fb202SetTestExecutionTimeout.bBusy) THEN
		fb202SetTestExecutionTimeout (bStart := FALSE);
		nStep := 0;
	END_IF
{endregion}
{endregion}
END_CASE

END_FUNCTION_BLOCK

// ---- POUs/DALI/PRGs/Diag/P_DALI_DIAG.TcPOU
PROGRAM P_DALI_DIAG
VAR
	fbDALIDiag: ARRAY [1.. SH_Light.DALI_Param.MAX_DALIV2_LINES] OF FB_DALI_Diag;
	bOneDaliBallastMissing: ARRAY [1.. SH_Light.DALI_Param.MAX_DALIV2_LINES] OF BOOL;
	bMissingShortAddress: ARRAY [1.. SH_Light.DALI_Param.MAX_DALIV2_LINES] OF BOOL;
	bSeveralMissingShortAddress: ARRAY [1.. SH_Light.DALI_Param.MAX_DALIV2_LINES] OF BOOL;
	
	nDiagIdx: BYTE;
END_VAR

fbDALIDiag[1].ipDALICommunication := P_DALI_Background.arrfbKL6821Communication[1];
fbDALIDiag[2].ipDALICommunication := P_DALI_Background.arrfbKL6821Communication[2];
fbDALIDiag[3].ipDALICommunication := P_DALI_Background.arrfbKL6821Communication[3];
fbDALIDiag[4].ipDALICommunication := P_DALI_Background.arrfbKL6821Communication[4];
fbDALIDiag[5].ipDALICommunication := P_DALI_Background.arrfbKL6821Communication[5];



FOR nDiagIdx := 1 TO MAX_DALIV2_LINES DO
	fbDALIDiag[nDiagIdx](
		bReInit:= , 
		bErrorFromSystem:= , 
		DALI_LINE_NUM:= nDiagIdx, 
		bOneDaliBallastMissing =>bOneDaliBallastMissing[nDiagIdx], 
		bMissingShortAddress=> bMissingShortAddress[nDiagIdx], 
		bSeveralMissingShortAddress=> bSeveralMissingShortAddress[nDiagIdx], 
		bBusy=> , 
		nErrorId=> GVL_AHDataModbus.arrFB_DALIDiagErrorId[nDiagIdx], 
		bErr=> );

END_FOR

END_PROGRAM

// ---- POUs/DALI/PRGs/EnergyData/P_DALI_Energy_Line.TcPOU
(*
EnergyReporting reads ActiveEnergy (part 252) for all present ballasts on all (configured) DALI-lines where GVL_DALI.g_arrEnergyData[*DALI-line*,*ballast*].bHasEnergyData is TRUE.
Results are stored in GVL_DALI.g_arrEnergyData[*DALI-line*,*ballast*].fActiveEnergy. Energy Data for individual ballasts is NOT persistent.
The engergy sum per DALI-Line (Wh) and Total Energy (kWh) are persistent.

If bCheckActiveEnergy is TRUE, all present ballasts are queried for ActiveEnergy and bHasEnergyData is updated accordingly.
This will result in errors for any ballast that does not comply with part 252.
Errors will not be triggered for activations where bCheckActiveEnergy is FALSE.

After shutdown or download to PLC EnergyReporting is activated automatically internally with bCheckActiveEnergy set to TRUE

EnergyReporting is activated automatically at TOD 0:00, 6:00, 12:00, 18:00 (configurable)

NB:	The priority of commands are set to "middle" internally. Updating all lines will take a couple of minutes to finish, so be patient.
	Other critical commands on the DALI-lines take priotity.
	Add appropriate communication immediately after configuration of a new KL6821 terminal.
	That is, arrfbDALI_EnergyReporting[*DALI-Line*].ipDALICommunication := P_DALI_Background.arrfbKL6821Communication[*DALI-Line*];
*)


PROGRAM P_DALI_Energy_Line
VAR
	arrfbDALI_EnergyReporting	: ARRAY[1..SH_Light.DALI_Param.MAX_DALIV2_LINES] OF FB_DALI_EnergyReporting;
	fbDALI_EnergyDataManagement	: SH_Light.FB_DALI_EnergyDataManagement;
	nNumOfEnergyLines			: BYTE;
	bReadEnergyDataAllLines		: BOOL;
	bReportingDone				: BOOL;
	fbRTrig_ReportingDone		: R_TRIG;
	bRTrigReportingDone			: BOOL;
	
	//Task scheduling
	stLocalSystemTime 		: TIMESTRUCT;
	fbLocalSystemTime 		: FB_LocalSystemTime;
	bGetTime 				: BOOL := TRUE;
	tTimeOut 				: TIME := DEFAULT_ADS_TIMEOUT;
	bLocalSystemTimeValid	: BOOL;
	tzID       				: E_TimeZoneID := eTimeZoneID_Invalid;
	
	tdSystemTime			: TOD;
	btestTodCompare			: BOOL;
	
	
END_VAR
VAR CONSTANT
	tdMidnight						: TOD := TOD#0:0:0;
	tdMorning						: TOD := TOD#6:0:0;
	tdMidDay						: TOD := TOD#12:0:0;
	tdEvening						: TOD := TOD#18:0:0;
	tCheckDuration					: TIME:= T#5S;
	tdTestsum						: TOD := (tdMidnight + tCheckDuration);
END_VAR

VAR PERSISTENT
	arrDaliLineEnergySumWh				: ARRAY[1..SH_Light.DALI_Param.MAX_DALIV2_LINES] OF LREAL;
	fTotalEnergyWh						: LREAL;
	nMaxControlGearOperatingHours		: UINT;
END_VAR


arrfbDALI_EnergyReporting[1].ipDALICommunication := P_DALI_Background.arrfbKL6821Communication[1];
arrfbDALI_EnergyReporting[2].ipDALICommunication := P_DALI_Background.arrfbKL6821Communication[2];
arrfbDALI_EnergyReporting[3].ipDALICommunication := P_DALI_Background.arrfbKL6821Communication[3];
arrfbDALI_EnergyReporting[4].ipDALICommunication := P_DALI_Background.arrfbKL6821Communication[4];
arrfbDALI_EnergyReporting[5].ipDALICommunication := P_DALI_Background.arrfbKL6821Communication[5];
//arrfbDALI_EnergyReporting[6].ipDALICommunication := P_DALI_Background.arrfbKL6821Communication[6]; // for more update SH_Light.DALI_Param.MAX_DALIV2_LINES

nNumOfEnergyLines := 5;

fbLocalSystemTime(
	sNetID:= '', 
	bEnable:= bGetTime, 
	dwCycle:= 2, // cycle time (in seconds) , Synchronization  every 2 seconds.
	dwOpt:= 1, //Bit 0: If this is set, the Windows system time is additionally synchronized cyclically with the hardware clock (RTC) (corresponds to the function NT_SetTimeToRTCTime).
	tTimeout:= tTimeOut, 
	bValid=> bLocalSystemTimeValid, 
	systemTime=> stLocalSystemTime, 
	tzID=> tzID);
	
tdSystemTime := SYSTEMTIME_TO_TOD(systemTime := stLocalSystemTime);
IF	((tdSystemTime > tdMidnight AND tdSystemTime < (tdMidnight + tCheckDuration)) OR (tdSystemTime > tdMorning AND tdSystemTime < (tdMorning + tCheckDuration)) OR
	(tdSystemTime > tdMidDay AND tdSystemTime < (tdMidDay + tCheckDuration)) OR (tdSystemTime > tdEvening AND tdSystemTime < (tdEvening + tCheckDuration))) THEN
	bReadEnergyDataAllLines := TRUE;
END_IF

fbDALI_EnergyDataManagement(
	NumOfEnergyLines				:= nNumOfEnergyLines,
	bReadEnergyDataAllLines 		:= bReadEnergyDataAllLines,
	arrfbDALI_EnergyReporting		:= arrfbDALI_EnergyReporting,
	arrDaliLineEnergySum			:= arrDaliLineEnergySumWH,
	fTotalEnergyWh					:= fTotalEnergyWh,
	nMaxControlGearOperatingHours	:= nMaxControlGearOperatingHours,
	bReportingDone					=> bReportingDone
);
GVL_AHDataModbus.nTotalEnergy10kWh := TO_UINT(TRUNC(fTotalEnergyWh*EXPT(10,-4)));  //FB_DALI_EnergyDataManagement makes sure only positive values are returned. As so, conversion from REAL to UINT is appropriate
GVL_AHDataModbus.nMaxControlGearOperatingHours := nMaxControlGearOperatingHours;
(*fbRTrig_ReportingDone(CLK:=bReportingDone, Q=> bRTrigReportingDone);
IF bRTrigReportingDone THEN
	GVL_AHDataModbus.nTotalEnergyKWH := nTotalEnergykWh;
	GVL_AHDataModbus.nMaxControlGearOperatingHours := nMaxControlGearOperatingHours;
END_IF*)

END_PROGRAM

// ---- POUs/EnOcean/P_EnOcean.TcPOU
PROGRAM P_EnOcean
VAR
	fbKL6581			: FB_KL6581;
	stKL6581_in  AT %I* : KL6581_INPUT;
	stKL6581_out AT %Q*	: KL6581_OUTPUT;
	stKL6581			: STR_KL6581;
	bInitCom			: BOOL := TRUE;
	
	arrEnOcean_Search	: ARRAY [1..8] OF FB_EnOcean_Search;
	nSearchIdx			: BYTE;
	bSerach				: BOOL;
	arrDevices			: ARRAY [1..8] OF INT;
	arrID				: ARRAY [1..8, 0..255] OF DWORD;
	
		//Trykknapper Atrium
	fbAtriumNiveau_Tryk_PladeB				: FB_Rec_RPS_Switch;
	fbAtriumNiveau_Tryk_Sevice				: FB_Rec_RPS_Switch;			

	//Trykknapper på gange

	
	//Trykknapper i rum
    fbRum_2_145_Tryk						: FB_Rec_RPS_Switch;
 
    fbRum_3_155_Tryk	                    : FB_Rec_RPS_Switch;


END_VAR

VAR CONSTANT
	byNode_1: BYTE := 1;
	byNode_2: BYTE := 2;
	byNode_3: BYTE := 3;
	byNode_4: BYTE := 4;
	byNode_5: BYTE := 5;
	byNode_6: BYTE := 6;
	byNode_7: BYTE := 7;
	byNode_8: BYTE := 8;
END_VAR


(* Kommunikation mit der KL6581. *)
(* Communication with the KL6581. *)
fbKL6581(
	bInit			:= bInitCom,
	nIdx			:= 2,
	stKL6581_in		:= stKL6581_In,
	stKL6581_out	:= stKL6581_Out,
	bReady			=> ,
	bBusy			=> ,
	bError			=> ,
	iErrorID		=> ,
	str_KL6581		=> stKL6581);

GVL_AHDataModbus.EnOceanError	:= TO_UINT(fbKL6581.iErrorID);
(* Warten bis der Kommunikationsbaustein initialisiert wurde.*)
(* Wait until the communication function block has been initialized. *)
IF (NOT fbKL6581.bReady) THEN
	RETURN;
END_IF

FOR nSearchIdx:= 1 TO 8 DO
	arrEnOcean_Search[nSearchIdx](
		bStart:= TRUE, 
		str_KL6581:= stKL6581 , 
		byNode:= nSearchIdx, 
		bReceive=> , 
		iDevices=>arrDevices[nSearchIdx] , 
		ar_ID=> );
		
		MEMCPY(ADR(arrID[nSearchIdx,0]), ADR(arrEnOcean_Search[nSearchIdx].ar_ID), SIZEOF(arrEnOcean_Search[nSearchIdx].ar_ID)); 
END_FOR

//Gange



//RUM
 //
A_Rum_3_155();
A_Rum_2_145_1();


//AtriumNiveau
A_AtriumNiveau();

ACTION A_AtriumNiveau:
fbAtriumNiveau_Tryk_PladeB(
	str_KL6581:=stKL6581 , 
	byNode:=0, 
	dw_ID:= 16#0029B92D, 
	str_EnOceanSwitch=> GVL_EnOcean.strEnOceanSwitch_AtriumNiveau_PladeB,
	by_Node=> , 
	bReceive=> );
(*
fbAtriumNiveau_Tryk_Sevice(
	str_KL6581:=stKL6581 , 
	byNode:=0, 
	dw_ID:= 16#00FEE4FE87, 
	str_EnOceanSwitch=> GVL_EnOcean.strEnOceanSwitch_AtriumNiveau_Service, 
	by_Node=> , 
	bReceive=> );
*)
END_ACTION

ACTION A_Rum_2_145_1:
fbRum_2_145_Tryk(
	str_KL6581:=stKL6581 , 
	byNode:=2 , 
	dw_ID:= 16#0029B743, 
	str_EnOceanSwitch=> GVL_EnOcean.strEnOceanSwitch_Rum_2_145, 
	by_Node=> , 
	bReceive=> );
END_ACTION

ACTION A_Rum_3_155:
fbRum_3_155_Tryk(
	str_KL6581:=stKL6581 , 
	byNode:=2 , 
	dw_ID:= 16#0029ACF5, 
	str_EnOceanSwitch=> GVL_EnOcean.strEnOceanSwitch_Rum_3_155, 
	by_Node=> , 
	bReceive=> );
END_ACTION

END_PROGRAM

// ---- VISUs/MAIN.TcPOU
PROGRAM MAIN
VAR
	nAlive: INT;
	breset: BOOL;
	nDemoVariable : INT;
	nCX8200_State	AT %I*	: UINT;
END_VAR

VAR PERSISTENT
	nDemoVar_Persist: INT;
END_VAR

nAlive:= nAlive + 1;
GVL_AHDataModbus.nCX8200_State_MB := nCX8200_State;

P_SystemDK.M_nCyclic(bReset := breset );
P_DALI_DIAG();
DALI_Commissioning();
P_DALI_Energy_Line();
P_AHModbusComm();
P_DALI_Background();

//Gange
P_Gang_2_143A();
P_Gang_3_159A();
P_Gang_3_157();
P_Gang_7_153();
P_Rum_2_135();
P_Gang_Atrium();
//P_Gang_atrium();



//FoldeDøre
//P_Foldedoer_5_125();

//Rum
P_Rum_2_145();
P_Rum_3_155();
P_Rum_3_157A();
P_Rum_3_155();

//Trapper
P_Trappe_T2();
P_Trappe_T3();
//Testprogrammer
//P_DALI_Energy_Firmware_Test();

END_PROGRAM

// ---- POUs/Alle_Rum/Rum_Med_DALI_Pir/Rum_2_145/Visualization_5_352_1_1_1_1_1_2.TcVIS
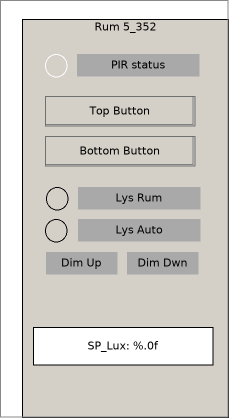
VISUALIZATION Visualization_5_352_1_1_1_1_1_2  // 229x418
    RoundedRectangle (22,19 207x399), "Rum 5_352"
    Rectangle (33,327 180x38), "SP_Lux: %.0f", text variable: P_Rum_4_324.fbLys.fbLightCtrl.fLuxZone1
    Button (45,96 150x30), "Top Button"
        tap P_Rum_5_352.bTopButtonZone1_Visu
    Button (45,136 150x30), "Bottom Button"
        tap P_Rum_5_352.bBottomButtonZone1_Visu
    Ellipse (46,187 22x23), colour toggle: P_Rum_5_352.fbLys.fbLightCtrl.bOnZone1
    Rectangle (78,187 122x22), "Lys Rum"
    Rectangle (46,252 71x22), "Dim Up", colour toggle: P_Rum_5_352.fbLys.fbLightCtrl.bDimUp
    Rectangle (127,252 71x22), "Dim Dwn", colour toggle: P_Rum_5_352.fbLys.fbLightCtrl.bDimDwn
    Ellipse (45,219 22x23), colour toggle: P_Rum_5_352.fbLys.fbLightCtrl.bAutoZone1
    Rectangle (78,219 122x22), "Lys Auto"
    Ellipse (45,54 22x23), colour toggle: P_Rum_5_352.fbLys.fbLightCtrl.bPIR
    Rectangle (77,54 122x22), "PIR status"
END_VISUALIZATION

// ---- POUs/Alle_Rum/Rum_Med_DALI_Pir/Rum_3_155/Visualization_5_352_1_1_1_1_1_2_1.TcVIS
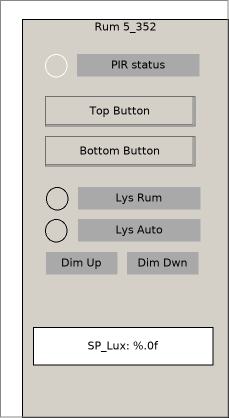
VISUALIZATION Visualization_5_352_1_1_1_1_1_2_1  // 229x418
    RoundedRectangle (22,19 207x399), "Rum 5_352"
    Rectangle (33,327 180x38), "SP_Lux: %.0f", text variable: P_Rum_4_324.fbLys.fbLightCtrl.fLuxZone1
    Button (45,96 150x30), "Top Button"
        tap P_Rum_5_352.bTopButtonZone1_Visu
    Button (45,136 150x30), "Bottom Button"
        tap P_Rum_5_352.bBottomButtonZone1_Visu
    Ellipse (46,187 22x23), colour toggle: P_Rum_5_352.fbLys.fbLightCtrl.bOnZone1
    Rectangle (78,187 122x22), "Lys Rum"
    Rectangle (46,252 71x22), "Dim Up", colour toggle: P_Rum_5_352.fbLys.fbLightCtrl.bDimUp
    Rectangle (127,252 71x22), "Dim Dwn", colour toggle: P_Rum_5_352.fbLys.fbLightCtrl.bDimDwn
    Ellipse (45,219 22x23), colour toggle: P_Rum_5_352.fbLys.fbLightCtrl.bAutoZone1
    Rectangle (78,219 122x22), "Lys Auto"
    Ellipse (45,54 22x23), colour toggle: P_Rum_5_352.fbLys.fbLightCtrl.bPIR
    Rectangle (77,54 122x22), "PIR status"
END_VISUALIZATION

// ---- POUs/Alle_Rum/Rum_Med_DALI_Pir/Rum_2_135/Visualization_5_352_1_1_1_1_1_2_1_1.TcVIS
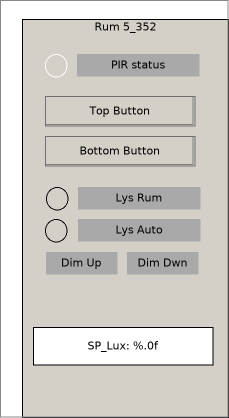
VISUALIZATION Visualization_5_352_1_1_1_1_1_2_1_1  // 229x418
    RoundedRectangle (22,19 207x399), "Rum 5_352"
    Rectangle (33,327 180x38), "SP_Lux: %.0f", text variable: P_Rum_4_324.fbLys.fbLightCtrl.fLuxZone1
    Button (45,96 150x30), "Top Button"
        tap P_Rum_5_352.bTopButtonZone1_Visu
    Button (45,136 150x30), "Bottom Button"
        tap P_Rum_5_352.bBottomButtonZone1_Visu
    Ellipse (46,187 22x23), colour toggle: P_Rum_5_352.fbLys.fbLightCtrl.bOnZone1
    Rectangle (78,187 122x22), "Lys Rum"
    Rectangle (46,252 71x22), "Dim Up", colour toggle: P_Rum_5_352.fbLys.fbLightCtrl.bDimUp
    Rectangle (127,252 71x22), "Dim Dwn", colour toggle: P_Rum_5_352.fbLys.fbLightCtrl.bDimDwn
    Ellipse (45,219 22x23), colour toggle: P_Rum_5_352.fbLys.fbLightCtrl.bAutoZone1
    Rectangle (78,219 122x22), "Lys Auto"
    Ellipse (45,54 22x23), colour toggle: P_Rum_5_352.fbLys.fbLightCtrl.bPIR
    Rectangle (77,54 122x22), "PIR status"
END_VISUALIZATION

// ---- POUs/DALI/DALI_Setup/VISUs/TextLists/ExtendedFadeTime.TcTLO
TEXTLIST ExtendedFadeTime
  0 = 'No Fade'
  1 = '1 * 100 ms = 100 ms'
  2 = '2 * 100 ms = 200 ms'
  3 = '3 * 100 ms = 300 ms'
  4 = '4 * 100 ms = 400 ms'
  5 = '5 * 100 ms = 500 ms'
  6 = '6 * 100 ms = 600 ms'
  7 = '7 * 100 ms = 700 ms'
  8 = '8 * 100 ms = 800 ms'
  9 = '9 * 100 ms = 900 ms'
  10 = '10 * 100 ms = 1000 ms'
  11 = '11 * 100 ms = 1100 ms'
  12 = '12 * 100 ms = 1200 ms'
  13 = '13 * 100 ms = 1300 ms'
  14 = '14 * 100 ms = 1400 ms'
  15 = '15 * 100 ms = 1500 ms'
  16 = '16 * 100 ms = 1600 ms'
  17 = '1 * 1 s = 1 s'
  18 = '2 * 1 s = 2 s'
  19 = '3 * 1 s = 3 s'
  20 = '4 * 1 s = 4 s'
  21 = '5 * 1 s = 5 s'
  22 = '6 * 1 s = 6 s'
  23 = '7 * 1 s = 7 s'
  24 = '8 * 1 s = 8 s'
  25 = '9 * 1 s = 9 s'
  26 = '10 * 1 s = 10 s'
  27 = '11 * 1 s = 11 s'
  28 = '12 * 1 s = 12 s'
  29 = '13 * 1 s = 13 s'
  30 = '14 * 1 s = 14 s'
  31 = '15 * 1 s = 15 s'
  32 = '16 * 1 s = 16 s'
  33 = '1 * 10 s = 10 s'
  34 = '2 * 10 s = 20 s'
  35 = '3 * 10 s = 30 s'
  36 = '4 * 10 s = 40 s'
  37 = '5 * 10 s = 50 s'
  38 = '6 * 10 s = 60 s'
  39 = '7 * 10 s = 70 s'
  40 = '8 * 10 s = 80 s'
  41 = '9 * 10 s = 90 s'
  42 = '10 * 10 s = 100 s'
  43 = '11 * 10 s = 110 s'
  44 = '12 * 10 s = 120 s'
  45 = '13 * 10 s = 130 s'
  46 = '14 * 10 s = 140 s'
  47 = '15 * 10 s = 150 s'
  48 = '16 * 10 s = 160 s'
  49 = '1 * 1 min = 1 min'
  50 = '2 * 1 min = 2 min'
  51 = '3 * 1 min = 3 min'
  52 = '4 * 1 min = 4 min'
  53 = '5 * 1 min = 5 min'
  54 = '6 * 1 min = 6 min'
  55 = '7 * 1 min = 7 min'
  56 = '8 * 1 min = 8 min'
  57 = '9 * 1 min = 9 min'
  58 = '10 * 1 min = 10 min'
  59 = '11 * 1 min = 11 min'
  60 = '12 * 1 min = 12 min'
  61 = '13 * 1 min = 13 min'
  62 = '14 * 1 min = 14 min'
  63 = '15 * 1 min = 15 min'
  64 = '16 * 1 min = 16 min'
  255 = 'Unknown'
   = ''
END_TEXTLIST

// ---- POUs/DALI/DALI_Setup/VISUs/Visu_DALICommissioning.TcVIS
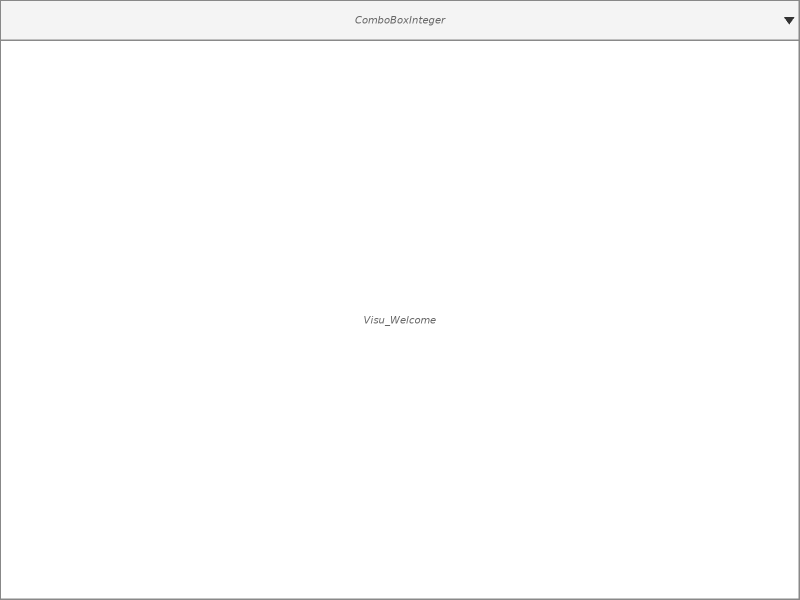
VISUALIZATION Visu_DALICommissioning  // 800x600
    ComboBoxInteger (0,0 800x40), variable: DALI_Commissioning.nSelectedDialog, input disabled if: DALI_Commissioning.bDisableComboBox, text list: 'TextList_Dialogs'
    Frame (0,40 800x560), frame switch variable: DALI_Commissioning.nSelectedDialog
        shows Visu_Welcome()
        shows Visu_Part102Commands()
        shows Visu_Part102Addressing()
        shows Visu_Part102Parameters()
        shows Visu_Part102Groups()
        shows Visu_Part102Scenes()
        shows Visu_Part102MemoryBank()
        shows Visu_Part102SetFading()
        shows Visu_Part202()
        shows Visu_Part205()
        shows Visu_Part207()
        shows Visu_Part208Switching()
        shows Visu_Part103Addressing()
        shows Visu_Part103Parameters()
        shows Visu_Part103Identify()
        shows Visu_Part301PushButton()
        shows Visu_Part302AbsoluteInputDevice()
        shows Visu_Part303OccupancySensor()
        shows Visu_Part304LightSensor()
        shows Visu_Part300GenericDevice()
        shows Visu_Part103MemoryBank()
        shows Visu_KL6821Configuration()
END_VISUALIZATION

// ---- POUs/DALI/DALI_Setup/VISUs/Visu_DALICommissioning/Visu_Part102MemoryBank.TcVIS
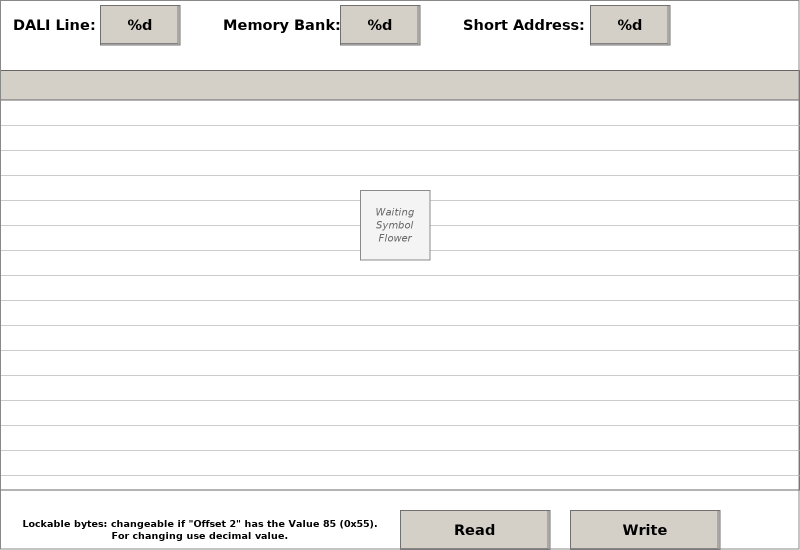
VISUALIZATION Visu_Part102MemoryBank  // 800x550
    Table (0,70 800x420), data array: DALI_Commissioning.fbPart102MemoryPages.aMemoryBank
        p1137915858: DALI_Commissioning.fbPart102MemoryPages.nOffset
        p3854506369: DALI_Commissioning.fbPart102MemoryPages.aMemoryBank[INDEX].sOffset
        p1892666644: DALI_Commissioning.fbPart102MemoryPages.aMemoryBank[INDEX].sName
        p338671338: DALI_Commissioning.fbPart102MemoryPages.aMemoryBank[INDEX].nValueDec
        p2170511999: DALI_Commissioning.fbPart102MemoryPages.aMemoryBank[INDEX].nValueHex
        p1755163831: Value Dec
        p4092479075: Value Hex
        Columns.Column.[0].Template: DALI_Commissioning.fbPart102MemoryPages.aNoValue[INDEX]
        Columns.Column.[1].Template: DALI_Commissioning.fbPart102MemoryPages.aNoValue[INDEX]
        Columns.Column.[2].Template: DALI_Commissioning.fbPart102MemoryPages.aNoValue[INDEX]; OnMouseClick: write the text variable via Default, min 0, max 255, title "Lockable variable decimal"
        Columns.Column.[3].Template: DALI_Commissioning.fbPart102MemoryPages.aNoValue[INDEX]; OnMouseClick: write the text variable via Default, title "Lockable variable hexadecimal"
    Button (400,510 150x40), "Read"
        OnMouseClick: execute { DALI_Commissioning.fbPart102MemoryPages.bRead := TRUE; }
    Button (570,510 150x40), "Write"
        OnMouseClick: execute { DALI_Commissioning.fbPart102MemoryPages.bWrite := TRUE; }
    Textfield (15,510 370x40), "Lockable bytes: changeable if "Offset 2" has the Value 85 (0x55). For changing use decimal value."
    WaitingSymbolFlower (360,190 70x70), invisible if: DALI_Commissioning.fbPart102MemoryPages.bHideWaitSymbol
    Textfield (460,5 130x40), "Short Address:"
    Button (590,5 80x40), "%d", text variable: DALI_Commissioning.fbPart102MemoryPages.nAddress
        OnMouseClick: write the text variable via Default, min 0, max 63, title "Insert Short Address"
    Textfield (220,5 120x40), "Memory Bank:"
    Button (340,5 80x40), "%d", text variable: DALI_Commissioning.fbPart102MemoryPages.nMemoryBank
        OnMouseClick: write the text variable via Default, min 0, max 255, title "Insert Memory Bank"
    Group (10,5 170x40)
        Textfield (0,0 110x40), "DALI Line:"
        Button (90,0 80x40), "%d", text variable: GVL_Internal.nDALILine
            OnMouseClick: write the text variable via Default, min 1, max 10, title "Choose line"
END_VISUALIZATION

// ---- POUs/DALI/DALI_Setup/VISUs/Visu_DALICommissioning/Visu_Part205Status.TcVIS
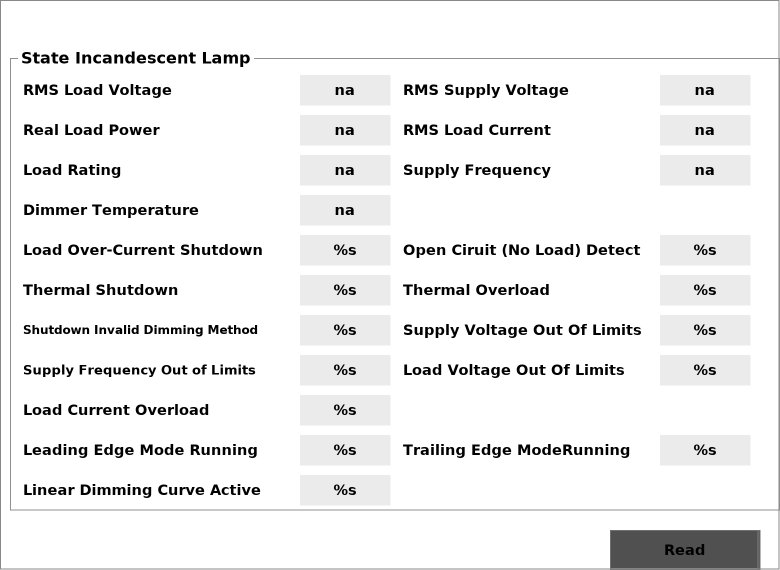
VISUALIZATION Visu_Part205Status  // 780x570
    Button (610,530 150x40), "Read"
        OnMouseClick: execute { DALI_Commissioning.fbPart205Incandescent.bReadStatus := TRUE; }
    GroupBox (10,50 770x460), "State Incandescent Lamp"
        Textfield (290,185 90x30), "%s", text variable: DALI_Commissioning.fbPart205Incandescent.sLoadOverCurrentShutdown
        Textfield (650,105 90x30), "%d Hz", text variable: DALI_Commissioning.fbPart205Incandescent.nSupplyFrequency
        Textfield (650,65 90x30), "%d %%", text variable: DALI_Commissioning.fbPart205Incandescent.nRMSLoadCurrent
        Textfield (650,25 90x30), "%d V", text variable: DALI_Commissioning.fbPart205Incandescent.nRMSSupplyVoltage
        Textfield (290,145 90x30), "%d °C", text variable: DALI_Commissioning.fbPart205Incandescent.nDimmerTemperature
        Textfield (290,105 90x30), "%2.1f mA", text variable: DALI_Commissioning.fbPart205Incandescent.fLoadRating
        Textfield (290,65 90x30), "%5.1f W", text variable: DALI_Commissioning.fbPart205Incandescent.fRealLoadPower
        Textfield (290,25 90x30), "%d V", text variable: DALI_Commissioning.fbPart205Incandescent.nRmsLoadVoltage
        Textfield (10,25 240x30), "RMS Load Voltage"
        Textfield (10,65 240x30), "Real Load Power", text variable: DALI_Commissioning.fbPart202Emergency.fFunctionTestDelayTimeVisu
        Textfield (10,145 240x30), "Dimmer Temperature"
        Textfield (10,105 240x30), "Load Rating"
        Textfield (10,185 240x30), "Load Over-Current Shutdown"
        Textfield (10,225 240x30), "Thermal Shutdown"
        Textfield (10,265 240x30), "Shutdown Invalid Dimming Method"
        Textfield (10,305 240x30), "Supply Frequency Out of Limits"
        Textfield (10,345 240x30), "Load Current Overload"
        Textfield (10,385 240x30), "Leading Edge Mode Running"
        Textfield (10,425 240x30), "Linear Dimming Curve Active"
        Textfield (290,265 90x30), "%s", text variable: DALI_Commissioning.fbPart205Incandescent.sInvalidDimmingMethod
        Textfield (290,305 90x30), "%s", text variable: DALI_Commissioning.fbPart205Incandescent.sSupplyFrequencyOutOfLimit
        Textfield (650,185 90x30), "%s", text variable: DALI_Commissioning.fbPart205Incandescent.sOpenCircuitDetection
        Textfield (650,225 90x30), "%s", text variable: DALI_Commissioning.fbPart205Incandescent.sThermalOverload
        Textfield (650,265 90x30), "%s", text variable: DALI_Commissioning.fbPart205Incandescent.sSupplyVoltageOutOfLimit
        Textfield (650,385 90x30), "%s", text variable: DALI_Commissioning.fbPart205Incandescent.sTrailingEdgeModeRunning
        Textfield (290,345 90x30), "%s", text variable: DALI_Commissioning.fbPart205Incandescent.sLoadCurrentOverload
        Textfield (290,385 90x30), "%s", text variable: DALI_Commissioning.fbPart205Incandescent.sLeadingEdgeModeRunning
        Textfield (290,425 90x30), "%s", text variable: DALI_Commissioning.fbPart205Incandescent.sLinearDimmingCurve
        Textfield (290,225 90x30), "%s", text variable: DALI_Commissioning.fbPart205Incandescent.sThermalShutdown
        Textfield (390,25 240x30), "RMS Supply Voltage"
        Textfield (390,65 240x30), "RMS Load Current"
        Textfield (390,105 240x30), "Supply Frequency"
        Textfield (390,185 240x30), "Open Ciruit (No Load) Detect"
        Textfield (390,225 240x30), "Thermal Overload"
        Textfield (390,265 240x30), "Supply Voltage Out Of Limits"
        Textfield (390,305 240x30), "Load Voltage Out Of Limits"
        Textfield (390,385 240x30), "Trailing Edge ModeRunning"
        Textfield (650,305 90x30), "%s", text variable: DALI_Commissioning.fbPart205Incandescent.sLoadVoltageOutOfLimit
        Textfield (290,25 90x30), "na", invisible if: not DALI_Commissioning.fbPart205Incandescent.bNoRmsLoadVoltage, input disabled if: true
        Textfield (290,65 90x30), "na", invisible if: not DALI_Commissioning.fbPart205Incandescent.bNoRealLoadPower, input disabled if: true
        Textfield (290,105 90x30), "na", invisible if: not DALI_Commissioning.fbPart205Incandescent.bNoLoadRating, input disabled if: true
        Textfield (290,145 90x30), "na", invisible if: not DALI_Commissioning.fbPart205Incandescent.bNoDimmerTemperature, input disabled if: true
        Textfield (650,25 90x30), "na", invisible if: not DALI_Commissioning.fbPart205Incandescent.bNoRMSSupplyVoltage, input disabled if: true
        Textfield (650,65 90x30), "na", invisible if: not DALI_Commissioning.fbPart205Incandescent.bNoRMSLoadCurrent, input disabled if: true
        Textfield (650,105 90x30), "na", invisible if: not DALI_Commissioning.fbPart205Incandescent.bNoSupplyFrequency, input disabled if: true
END_VISUALIZATION
